// TIA Portal V20 export
TYPE "LConSMC_typeTechnollogyControllerDiag"
// Diagnosedaten des Technologiereglers / Diagnostic data of the technology controller
// stored: Access Published
   STRUCT
      pidoutValue : LReal := 0.0;   // PID-Regler Ausgang: Drehmomentenregelung [N oder Lbf] Geschwindigkeitsadaption [m/min or ft/min] / PID-controller output value: Torque control [N or Lbf] Velocity adaption [m/min or ft/min]
      pidEffectiveKp : LReal := 0.0;   // Effektive P-Verstärkung wenn die Adaption verwendet wird / Effective P-gain if the gain adaption is used
      pidUpperLimitReached : Bool := FALSE;   // TRUE: PID Ausgang hat die untere Grenze erreicht / TRUE: PID output has reached the upper limit
      pidLowerLimitReached : Bool := FALSE;   // TRUE: PID Ausgang hat die obere Grenze erreicht / TRUE: PID output has reached the upper limit
      pidRFGSetpointReached : Bool := FALSE;   // TRUE: Der interne Hochlaufgeber hat auf den Sollwert gerampt / TRUE: The internal ramp generator has reached the setpoint
   END_STRUCT;
END_TYPE
